ABB RobotStudio station: Assistenzsystem für Verpressung.rsstnx

Station Assistenzsystem für Verpressung (saved by RobotStudio 22.3.10190.2)
Controller IRB14000
  mechanical unit ROB_R: IRB14000_0.5_0.5_R, 6 joints, base frame (0, 0, 0) mm
  mechanical unit ROB_R_7: IRB14000_0.5_0.5_R, 1 joints, base frame (0, 0, 0) mm
  mechanical unit ROB_L: IRB14000_0.5_0.5_L, 6 joints, base frame (0, 0, 0) mm
  mechanical unit ROB_L_7: IRB14000_0.5_0.5_L, 1 joints, base frame (0, 0, 0) mm
Layout (positions relative to the parent item):
  - IRB14000_0.5_0.5 [mechanism, from Robots\IRB14000_0.5_0.5__01.rslib] at (0, 0, 0) mm
  - IRB14000_0.5_0.5_R [mechanism, from Robots\IRB14000_0.5_0.5__01.rslib] at (0, 0, 0) mm; joint values [0.3584, -1.8727, -2.4697, 0.5522, 0.721, 0.9332, -0.6165] (rad or m)
  - IRB14000_0.5_0.5_L [mechanism, from Robots\IRB14000_0.5_0.5__01.rslib] at (0, 0, 0) mm; joint values [-0.3584, -1.8727, 2.4697, 0.5522, -0.721, 0.9332, 0.6165] (rad or m)
